Xinje XCPPro project, PLC1: XC3-24 (software 3.3m)

PROGRAM Ladder

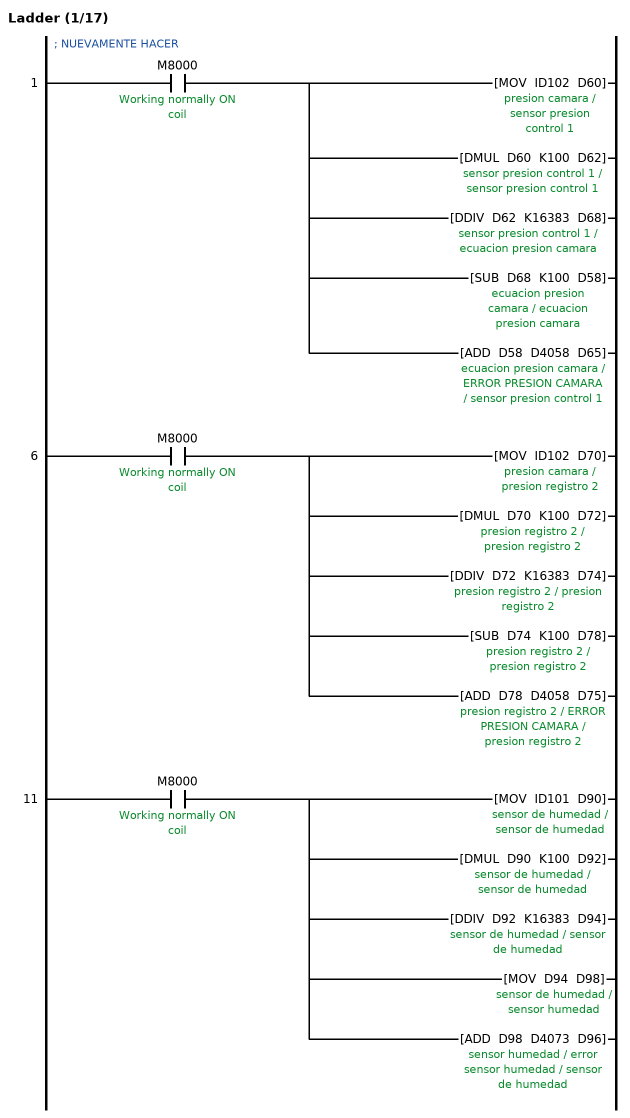
;  NUEVAMENTE HACER
LD     M8000	; Working normally ON coil
MOV    ID102 D60	; presion camara / sensor presion control 1
DMUL   D60 K100 D62	; sensor presion control 1 / sensor presion control 1
DDIV   D62 K16383 D68	; sensor presion control 1 / ecuacion presion camara
SUB    D68 K100 D58	; ecuacion presion camara / ecuacion presion camara
ADD    D58 D4058 D65	; ecuacion presion camara / ERROR PRESION CAMARA / sensor presion control 1
LD     M8000	; Working normally ON coil
MOV    ID102 D70	; presion camara / presion registro 2
DMUL   D70 K100 D72	; presion registro 2 / presion registro 2
DDIV   D72 K16383 D74	; presion registro 2 / presion registro 2
SUB    D74 K100 D78	; presion registro 2 / presion registro 2
ADD    D78 D4058 D75	; presion registro 2 / ERROR PRESION CAMARA / presion registro 2
LD     M8000	; Working normally ON coil
MOV    ID101 D90	; sensor de humedad / sensor de humedad
DMUL   D90 K100 D92	; sensor de humedad / sensor de humedad
DDIV   D92 K16383 D94	; sensor de humedad / sensor de humedad
MOV    D94 D98	; sensor de humedad / sensor humedad
ADD    D98 D4073 D96	; sensor humedad / error sensor humedad / sensor de humedad

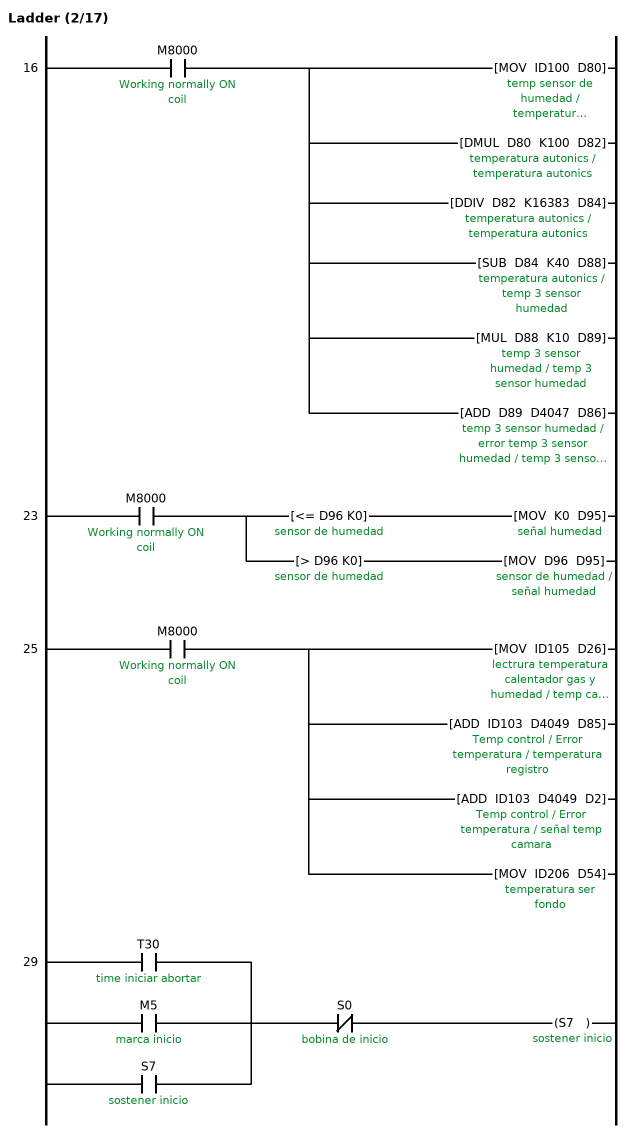
LD     M8000	; Working normally ON coil
MOV    ID100 D80	; temp sensor de humedad / temperatura autonics
DMUL   D80 K100 D82	; temperatura autonics / temperatura autonics
DDIV   D82 K16383 D84	; temperatura autonics / temperatura autonics
SUB    D84 K40 D88	; temperatura autonics / temp 3 sensor humedad
MUL    D88 K10 D89	; temp 3 sensor humedad / temp 3 sensor humedad
ADD    D89 D4047 D86	; temp 3 sensor humedad / error temp 3 sensor humedad / temp 3 sensor humedad
LD     M8000	; Working normally ON coil
MPS
AND<=  D96 K0	; sensor de humedad
MOV    K0 D95	; señal humedad
MPP
AND>   D96 K0	; sensor de humedad
MOV    D96 D95	; sensor de humedad / señal humedad
LD     M8000	; Working normally ON coil
MOV    ID105 D26	; lectrura temperatura  calentador gas y humedad / temp cal gas
ADD    ID103 D4049 D85	; Temp control / Error temperatura / temperatura registro
ADD    ID103 D4049 D2	; Temp control / Error temperatura / señal temp camara
MOV    ID206 D54	; temperatura ser fondo
LD     T30	; time iniciar abortar
OR     M5	; marca inicio
OR     S7	; sostener inicio
ANI    S0	; bobina de inicio
OUT    S7	; sostener inicio

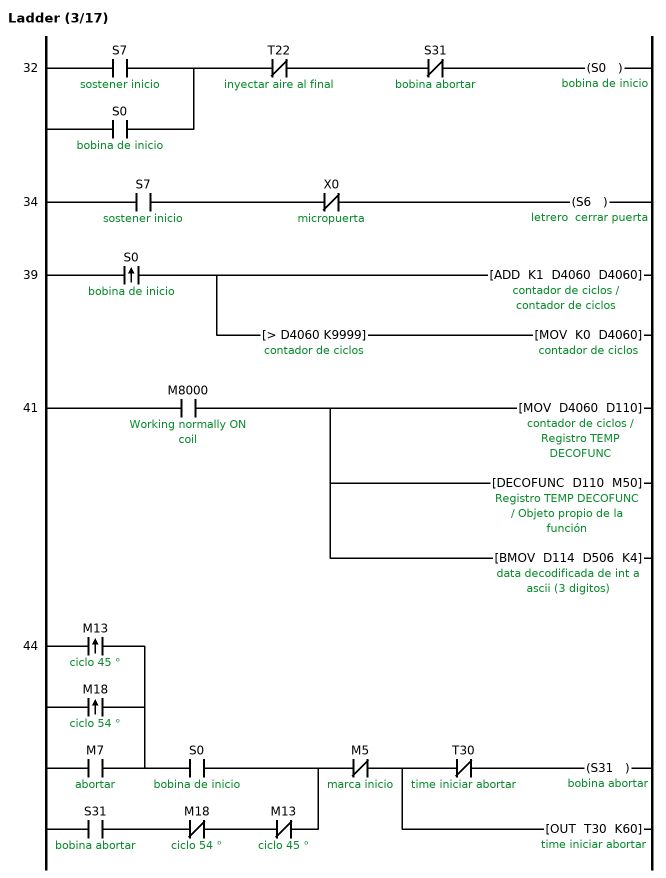
LD     S7	; sostener inicio
OR     S0	; bobina de inicio
ANI    T22	; inyectar aire al final
ANI    S31	; bobina abortar
OUT    S0	; bobina de inicio
LD     S7	; sostener inicio
ANI    X0	;  micropuerta
OUT    S6	; letrero  cerrar puerta
LDP    S0	; bobina de inicio
ADD    K1 D4060 D4060	; contador de ciclos / contador de ciclos
AND>   D4060 K9999	; contador de ciclos
MOV    K0 D4060	; contador de ciclos
LD     M8000	; Working normally ON coil
MOV    D4060 D110	; contador de ciclos / Registro TEMP DECOFUNC
DECOFUNC D110 M50	; Registro TEMP DECOFUNC / Objeto propio de la función
BMOV   D114 D506 K4	; data decodificada de int a ascii (3 digitos)
LDP    M13	; ciclo 45 °
ORP    M18	; ciclo 54 °
OR     M7	; abortar
AND    S0	; bobina de inicio
LD     S31	; bobina abortar
ANI    M18	; ciclo 54 °
ANI    M13	; ciclo 45 °
ORB
ANI    M5	; marca inicio
MPS
ANI    T30	; time iniciar abortar
OUT    S31	; bobina abortar
MPP
OUT    T30 K60	; time iniciar abortar

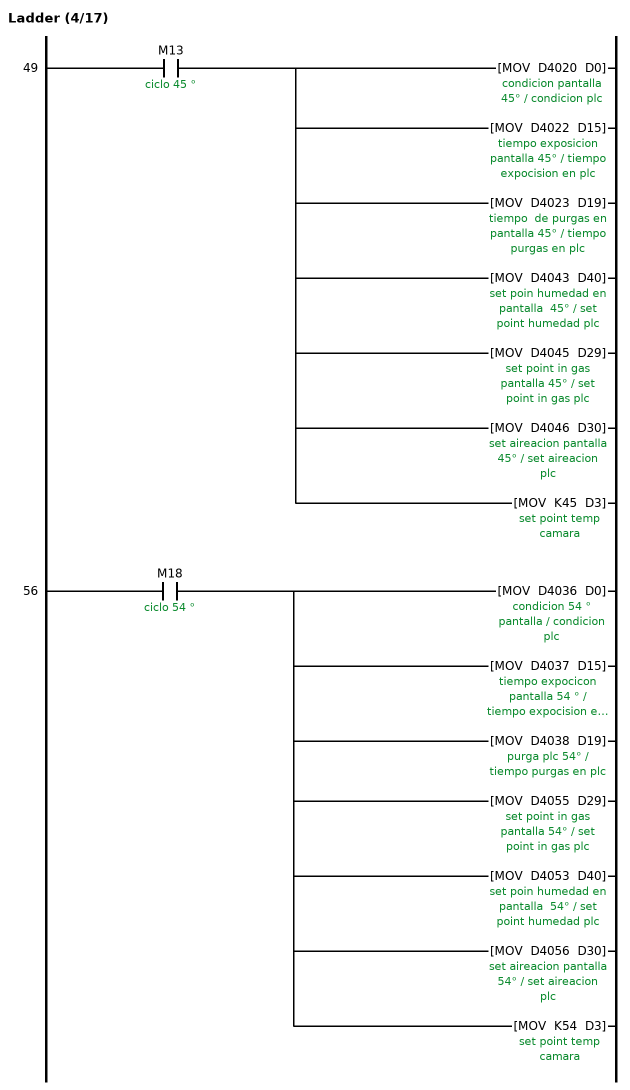
LD     M13	; ciclo 45 °
MOV    D4020 D0	; condicion pantalla 45° / condicion plc
MOV    D4022 D15	; tiempo exposicion pantalla 45° / tiempo expocision en plc
MOV    D4023 D19	; tiempo  de purgas en pantalla 45° / tiempo purgas en plc
MOV    D4043 D40	; set poin humedad en pantalla  45° / set point humedad plc
MOV    D4045 D29	; set point in gas  pantalla 45° / set point in gas plc
MOV    D4046 D30	; set aireacion pantalla 45° / set aireacion plc
MOV    K45 D3	; set point temp camara
LD     M18	; ciclo 54 °
MOV    D4036 D0	; condicion 54 ° pantalla / condicion plc
MOV    D4037 D15	; tiempo expocicon pantalla 54 ° / tiempo expocision en plc
MOV    D4038 D19	; purga plc 54° / tiempo purgas en plc
MOV    D4055 D29	; set point in gas  pantalla 54° / set point in gas plc
MOV    D4053 D40	; set poin humedad en pantalla  54° / set point humedad plc
MOV    D4056 D30	; set aireacion pantalla 54° / set aireacion plc
MOV    K54 D3	; set point temp camara

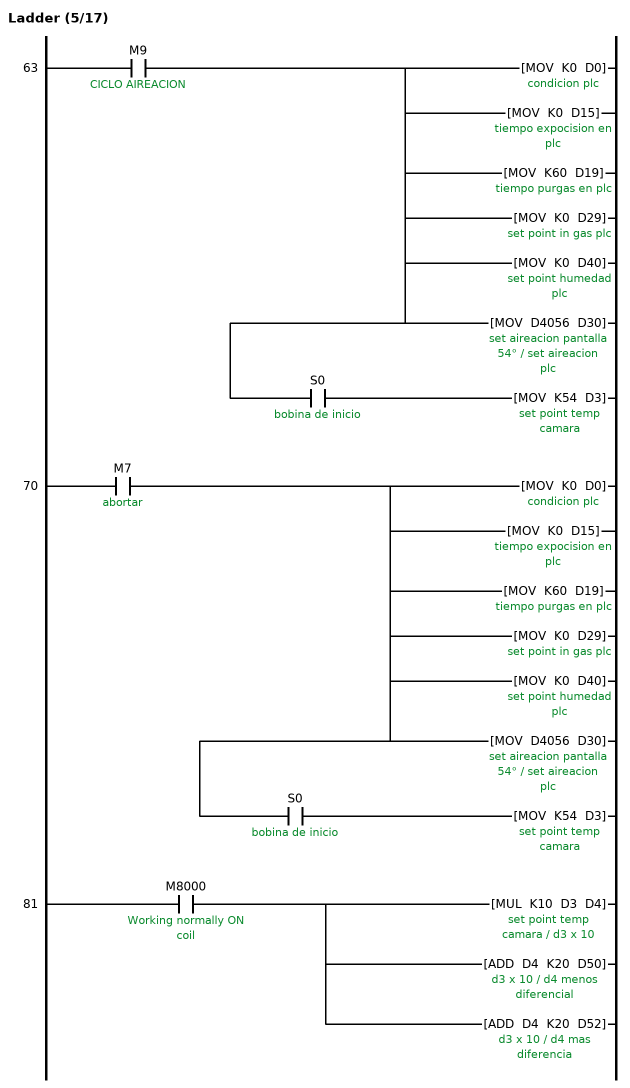
LD     M9	; CICLO AIREACION
MOV    K0 D0	; condicion plc
MOV    K0 D15	; tiempo expocision en plc
MOV    K60 D19	; tiempo purgas en plc
MOV    K0 D29	; set point in gas plc
MOV    K0 D40	; set point humedad plc
MOV    D4056 D30	; set aireacion pantalla 54° / set aireacion plc
AND    S0	; bobina de inicio
MOV    K54 D3	; set point temp camara
LD     M7	; abortar
MOV    K0 D0	; condicion plc
MOV    K0 D15	; tiempo expocision en plc
MOV    K60 D19	; tiempo purgas en plc
MOV    K0 D29	; set point in gas plc
MOV    K0 D40	; set point humedad plc
MOV    D4056 D30	; set aireacion pantalla 54° / set aireacion plc
AND    S0	; bobina de inicio
MOV    K54 D3	; set point temp camara
LD     M8000	; Working normally ON coil
MUL    K10 D3 D4	; set point temp camara / d3 x 10
ADD    D4 K20 D50	; d3 x 10 / d4 menos diferencial
ADD    D4 K20 D52	; d3 x 10 / d4 mas diferencia

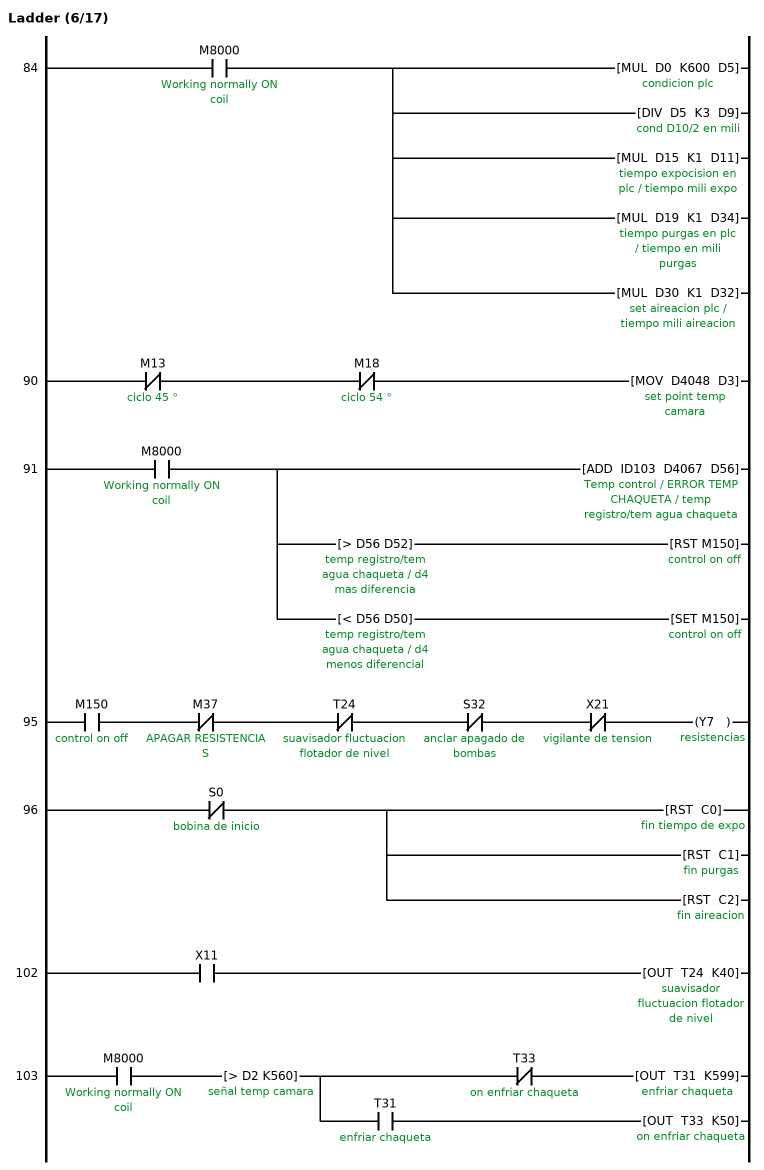
LD     M8000	; Working normally ON coil
MUL    D0 K600 D5	; condicion plc
DIV    D5 K3 D9	; cond D10/2 en mili
MUL    D15 K1 D11	; tiempo expocision en plc / tiempo mili expo
MUL    D19 K1 D34	; tiempo purgas en plc / tiempo en mili purgas
MUL    D30 K1 D32	; set aireacion plc / tiempo mili aireacion
LDI    M13	; ciclo 45 °
ANI    M18	; ciclo 54 °
MOV    D4048 D3	; set point temp camara
LD     M8000	; Working normally ON coil
ADD    ID103 D4067 D56	; Temp control / ERROR TEMP CHAQUETA / temp registro/tem agua chaqueta
MPS
AND>   D56 D52	; temp registro/tem agua chaqueta / d4 mas diferencia
RST    M150	; control on off
MPP
AND<   D56 D50	; temp registro/tem agua chaqueta / d4 menos diferencial
SET    M150	; control on off
LD     M150	; control on off
ANI    M37	; APAGAR RESISTENCIAS
ANI    T24	; suavisador fluctuacion flotador de nivel
ANI    S32	; anclar apagado de bombas
ANI    X21	; vigilante de tension
OUT    Y7	; resistencias
LDI    S0	; bobina de inicio
RST    C0	; fin tiempo de expo
RST    C1	; fin purgas
RST    C2	; fin aireacion
LD     X11
OUT    T24 K40	; suavisador fluctuacion flotador de nivel
LD     M8000	; Working normally ON coil
AND>   D2 K560	; señal temp camara
MPS
ANI    T33	; on enfriar chaqueta
OUT    T31 K599	; enfriar chaqueta
MPP
AND    T31	; enfriar chaqueta
OUT    T33 K50	; on enfriar chaqueta

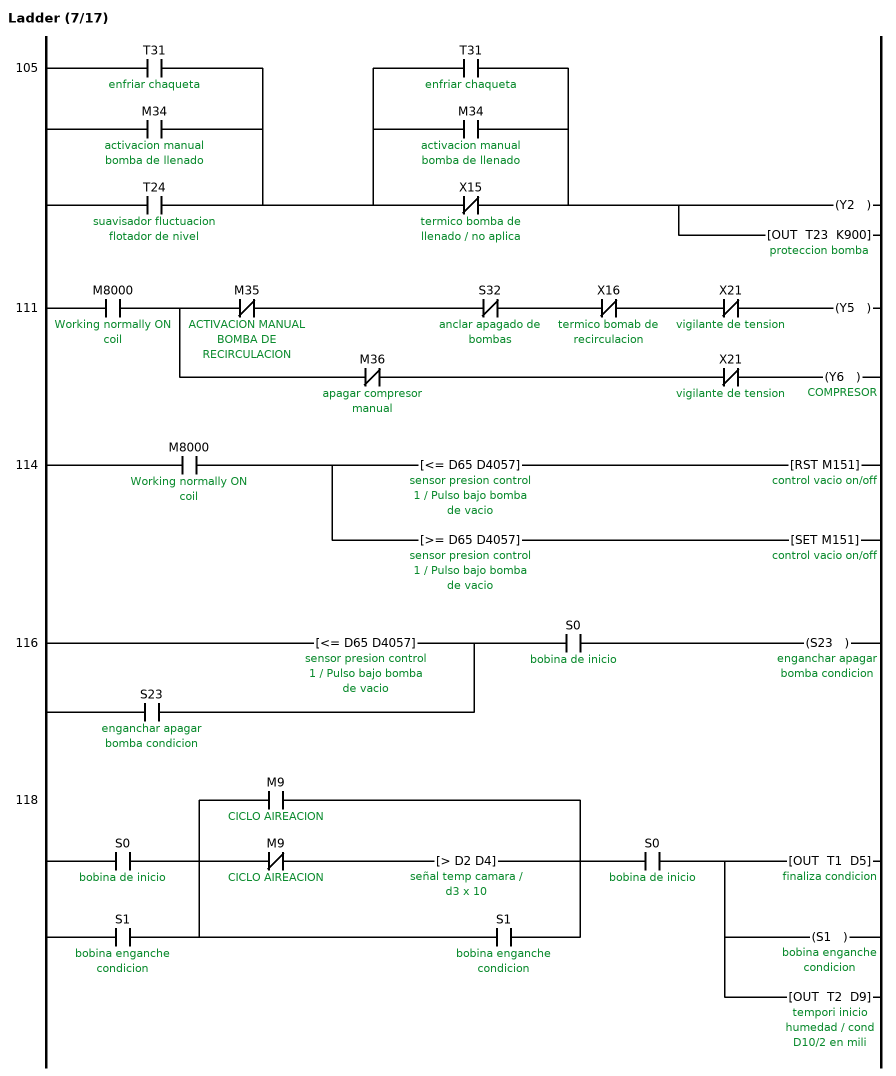
LD     T31	; enfriar chaqueta
OR     M34	; activacion manual bomba de llenado
OR     T24	; suavisador fluctuacion flotador de nivel
LD     T31	; enfriar chaqueta
OR     M34	; activacion manual bomba de llenado
ORI    X15	; termico bomba de  llenado / no aplica 
ANB
OUT    Y2
OUT    T23 K900	; proteccion bomba
LD     M8000	; Working normally ON coil
MPS
ANI    M35	; ACTIVACION MANUAL BOMBA DE RECIRCULACION
ANI    S32	; anclar apagado de bombas
ANI    X16	; termico bomab de recirculacion
ANI    X21	; vigilante de tension
OUT    Y5
MPP
ANI    M36	; apagar compresor manual
ANI    X21	; vigilante de tension
OUT    Y6	; COMPRESOR
LD     M8000	; Working normally ON coil
MPS
AND<=  D65 D4057	; sensor presion control 1 / Pulso bajo bomba de vacio
RST    M151	; control vacio on/off
MPP
AND>=  D65 D4057	; sensor presion control 1 / Pulso bajo bomba de vacio
SET    M151	; control vacio on/off
LD<=   D65 D4057	; sensor presion control 1 / Pulso bajo bomba de vacio
OR     S23	; enganchar apagar bomba condicion
AND    S0	; bobina de inicio
OUT    S23	; enganchar apagar bomba condicion
LD     S0	; bobina de inicio
OR     S1	; bobina enganche  condicion
LD     M9	; CICLO AIREACION
LDI    M9	; CICLO AIREACION
AND>   D2 D4	; señal temp camara / d3 x 10
ORB
OR     S1	; bobina enganche  condicion
ANB
AND    S0	; bobina de inicio
OUT    T1 D5	; finaliza condicion
OUT    S1	; bobina enganche  condicion
OUT    T2 D9	; tempori inicio humedad / cond D10/2 en mili

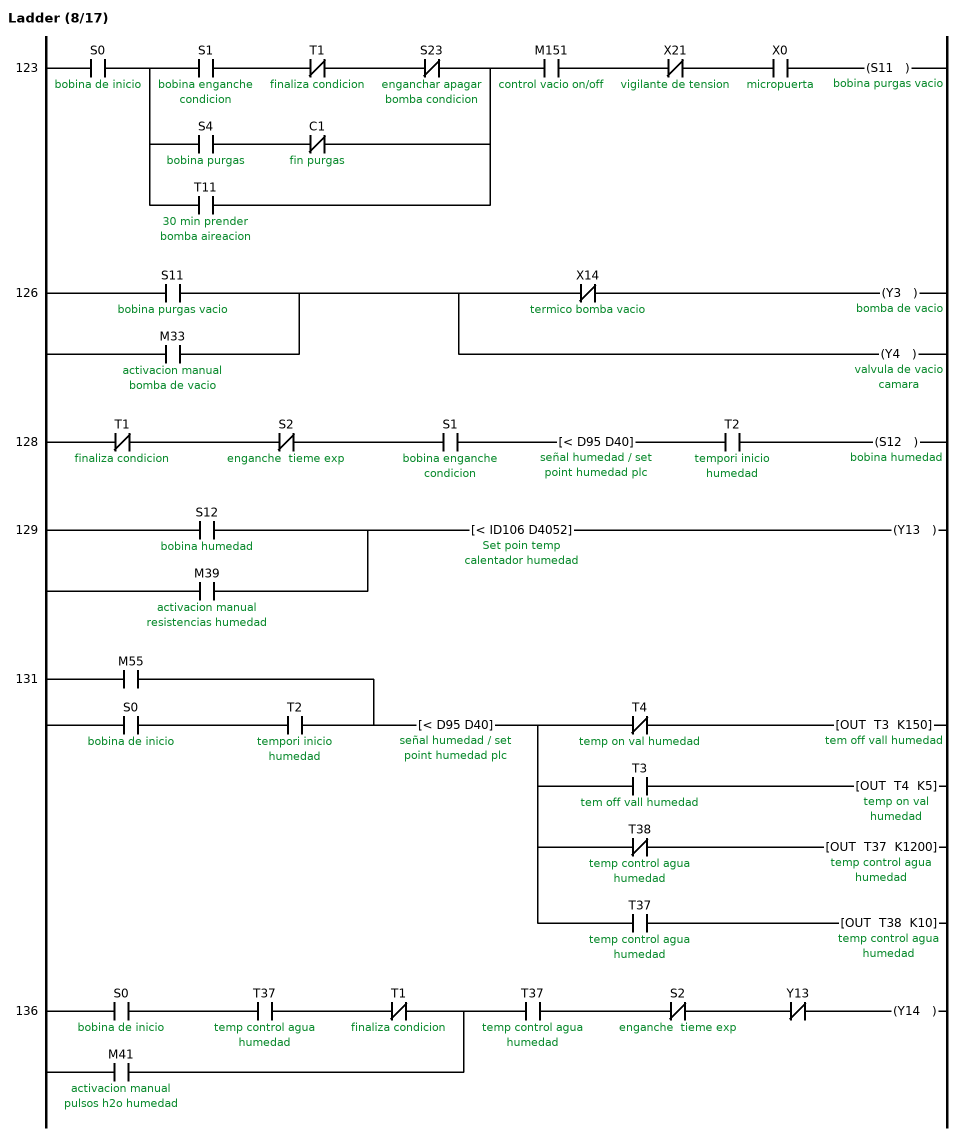
LD     S0	; bobina de inicio
LD     S1	; bobina enganche  condicion
ANI    T1	; finaliza condicion
ANI    S23	; enganchar apagar bomba condicion
LD     S4	; bobina purgas
ANI    C1	; fin purgas
ORB
OR     T11	; 30 min prender bomba aireacion
ANB
AND    M151	; control vacio on/off
ANI    X21	; vigilante de tension
AND    X0	;  micropuerta
OUT    S11	; bobina purgas vacio
LD     S11	; bobina purgas vacio
OR     M33	; activacion manual bomba de vacio
MPS
ANI    X14	; termico bomba vacio
OUT    Y3	; bomba de vacio
MPP
OUT    Y4	; valvula de vacio camara
LDI    T1	; finaliza condicion
ANI    S2	; enganche  tieme exp
AND    S1	; bobina enganche  condicion
AND<   D95 D40	; señal humedad / set point humedad plc
AND    T2	; tempori inicio humedad
OUT    S12	; bobina humedad
LD     S12	; bobina humedad
OR     M39	; activacion manual resistencias humedad
AND<   ID106 D4052	; Set poin temp calentador humedad
OUT    Y13
LD     M55
LD     S0	; bobina de inicio
AND    T2	; tempori inicio humedad
ORB
AND<   D95 D40	; señal humedad / set point humedad plc
MPS
ANI    T4	; temp on val humedad
OUT    T3 K150	; tem off vall humedad
MRD
AND    T3	; tem off vall humedad
OUT    T4 K5	; temp on val humedad
MRD
ANI    T38	; temp control agua humedad
OUT    T37 K1200	; temp control agua  humedad
MPP
AND    T37	; temp control agua  humedad
OUT    T38 K10	; temp control agua humedad
LD     S0	; bobina de inicio
AND    T37	; temp control agua  humedad
ANI    T1	; finaliza condicion
OR     M41	; activacion manual pulsos h2o humedad
AND    T37	; temp control agua  humedad
ANI    S2	; enganche  tieme exp
ANI    Y13
OUT    Y14

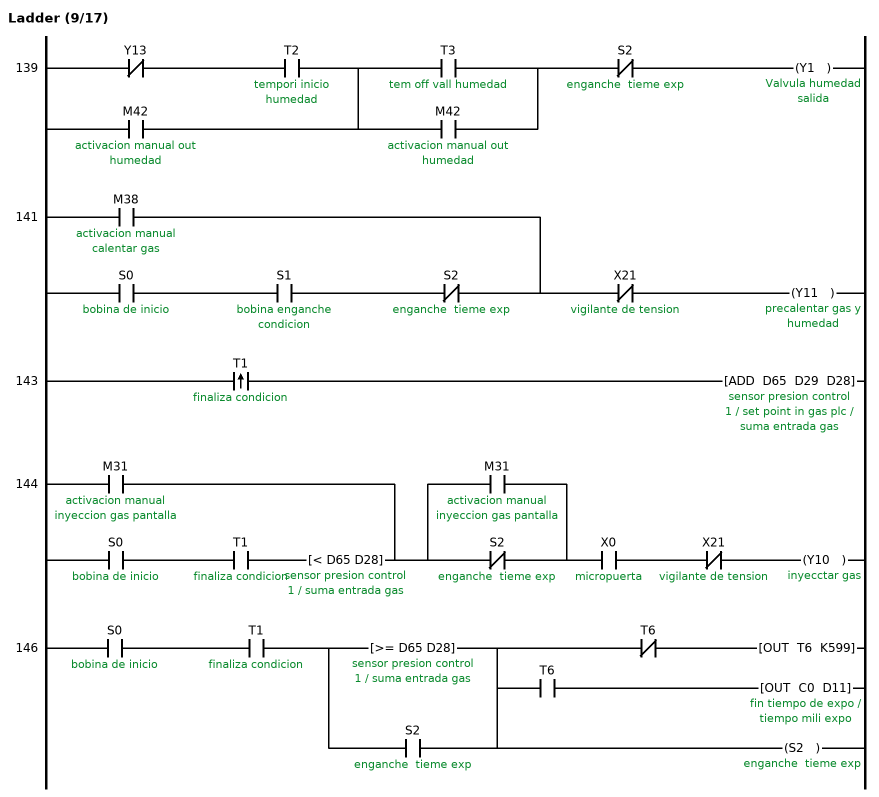
LDI    Y13
AND    T2	; tempori inicio humedad
OR     M42	; activacion manual out humedad
LD     T3	; tem off vall humedad
OR     M42	; activacion manual out humedad
ANB
ANI    S2	; enganche  tieme exp
OUT    Y1	; Valvula humedad salida
LD     M38	; activacion manual calentar gas
LD     S0	; bobina de inicio
AND    S1	; bobina enganche  condicion
ANI    S2	; enganche  tieme exp
ORB
ANI    X21	; vigilante de tension
OUT    Y11	; precalentar gas y humedad
LDP    T1	; finaliza condicion
ADD    D65 D29 D28	; sensor presion control 1 / set point in gas plc / suma entrada gas
LD     M31	; activacion manual inyeccion gas pantalla
LD     S0	; bobina de inicio
AND    T1	; finaliza condicion
AND<   D65 D28	; sensor presion control 1 / suma entrada gas
ORB
LD     M31	; activacion manual inyeccion gas pantalla
ORI    S2	; enganche  tieme exp
ANB
AND    X0	;  micropuerta
ANI    X21	; vigilante de tension
OUT    Y10	; inyecctar gas
LD     S0	; bobina de inicio
AND    T1	; finaliza condicion
LD>=   D65 D28	; sensor presion control 1 / suma entrada gas
OR     S2	; enganche  tieme exp
ANB
MPS
ANI    T6
OUT    T6 K599
MRD
AND    T6
OUT    C0 D11	; fin tiempo de expo / tiempo mili expo
MPP
OUT    S2	; enganche  tieme exp

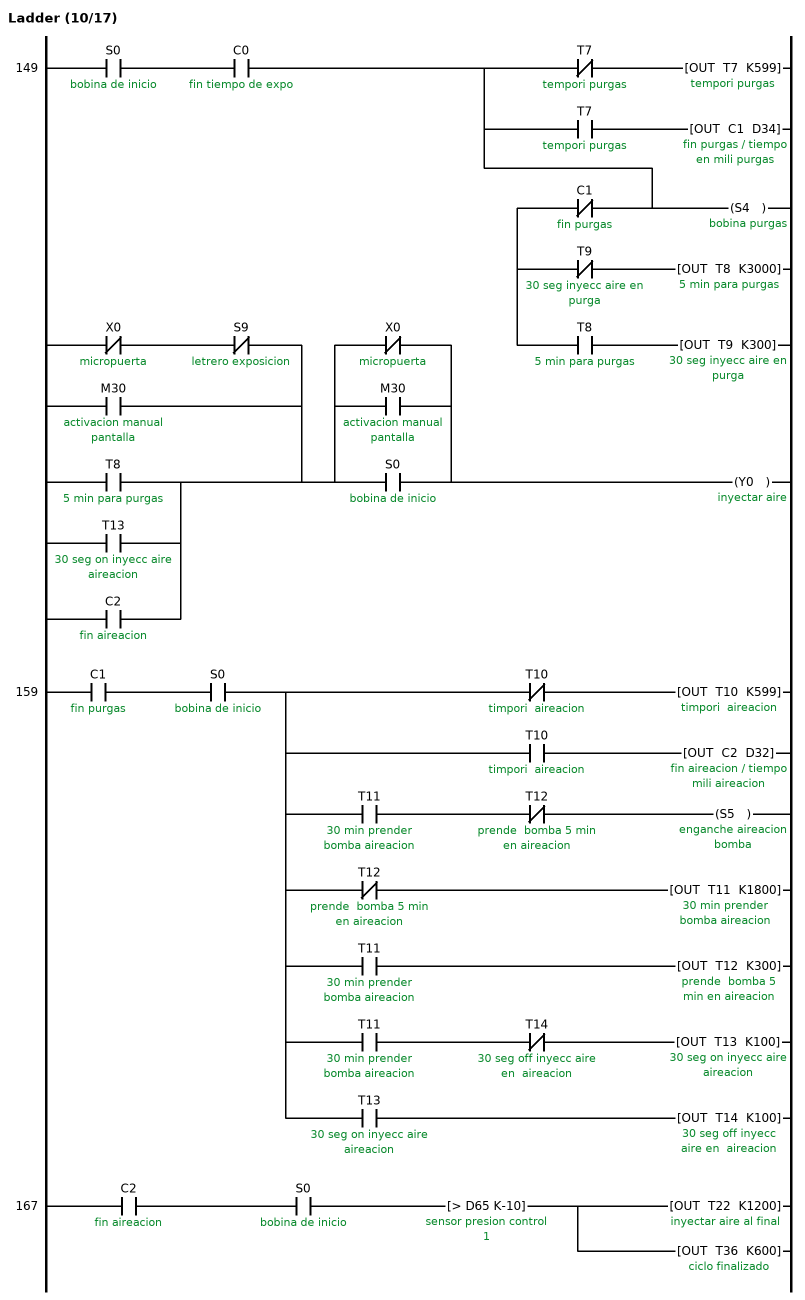
; (network is not series-parallel: see picture) LD S0 | LD C0 | LDI T7 | OUT T7 K599 | LD T7 | OUT C1 D34 | LDI C1 | OUT S4 | LDI T9 | OUT T8 K3000 | LDI X0 | LDI S9 | LDI X0 | LD T8 | OUT T9 K300 | LD M30 | LD M30 | LD T8 | LD S0 | OUT Y0 | LD T13 | LD C2
LD     C1	; fin purgas
AND    S0	; bobina de inicio
MPS
ANI    T10	; timpori  aireacion
OUT    T10 K599	; timpori  aireacion
MRD
AND    T10	; timpori  aireacion
OUT    C2 D32	; fin aireacion / tiempo mili aireacion
MRD
AND    T11	; 30 min prender bomba aireacion
ANI    T12	; prende  bomba 5 min en aireacion
OUT    S5	; enganche aireacion bomba
MRD
ANI    T12	; prende  bomba 5 min en aireacion
OUT    T11 K1800	; 30 min prender bomba aireacion
MRD
AND    T11	; 30 min prender bomba aireacion
OUT    T12 K300	; prende  bomba 5 min en aireacion
MRD
AND    T11	; 30 min prender bomba aireacion
ANI    T14	; 30 seg off inyecc aire en  aireacion
OUT    T13 K100	; 30 seg on inyecc aire aireacion
MPP
AND    T13	; 30 seg on inyecc aire aireacion
OUT    T14 K100	; 30 seg off inyecc aire en  aireacion
LD     C2	; fin aireacion
AND    S0	; bobina de inicio
AND>   D65 K-10	; sensor presion control 1
OUT    T22 K1200	; inyectar aire al final
OUT    T36 K600	; ciclo finalizado

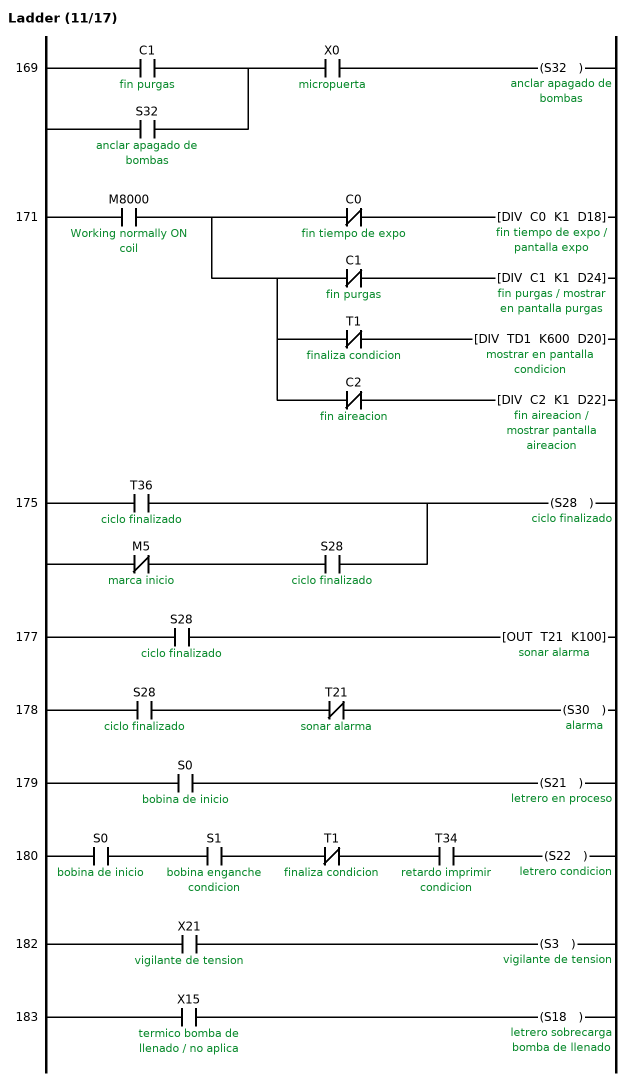
LD     C1	; fin purgas
OR     S32	; anclar apagado de bombas
AND    X0	;  micropuerta
OUT    S32	; anclar apagado de bombas
LD     M8000	; Working normally ON coil
MPS
ANI    C0	; fin tiempo de expo
DIV    C0 K1 D18	; fin tiempo de expo / pantalla expo
MRD
ANI    C1	; fin purgas
DIV    C1 K1 D24	; fin purgas / mostrar en pantalla purgas
MRD
ANI    T1	; finaliza condicion
DIV    TD1 K600 D20	; mostrar en pantalla condicion
MPP
ANI    C2	; fin aireacion
DIV    C2 K1 D22	; fin aireacion / mostrar pantalla aireacion
LD     T36	; ciclo finalizado
LDI    M5	; marca inicio
AND    S28	; ciclo finalizado
ORB
OUT    S28	; ciclo finalizado
LD     S28	; ciclo finalizado
OUT    T21 K100	; sonar alarma
LD     S28	; ciclo finalizado
ANI    T21	; sonar alarma
OUT    S30	; alarma
LD     S0	; bobina de inicio
OUT    S21	; letrero en proceso
LD     S0	; bobina de inicio
AND    S1	; bobina enganche  condicion
ANI    T1	; finaliza condicion
AND    T34	; retardo imprimir condicion
OUT    S22	; letrero condicion
LD     X21	; vigilante de tension
OUT    S3	; vigilante de tension
LD     X15	; termico bomba de  llenado / no aplica 
OUT    S18	; letrero sobrecarga bomba de llenado

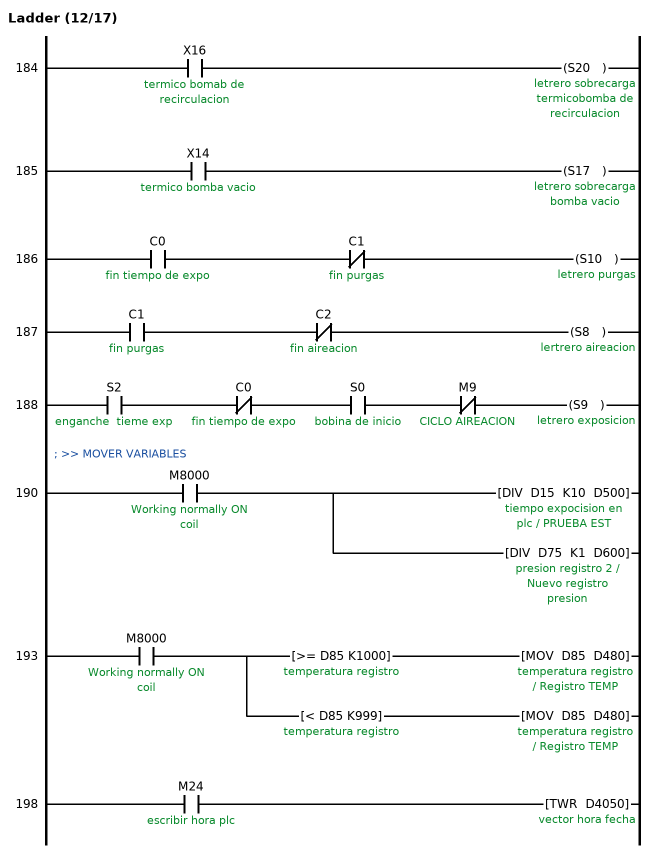
LD     X16	; termico bomab de recirculacion
OUT    S20	; letrero sobrecarga termicobomba de recirculacion
LD     X14	; termico bomba vacio
OUT    S17	; letrero sobrecarga bomba vacio
LD     C0	; fin tiempo de expo
ANI    C1	; fin purgas
OUT    S10	; letrero purgas
LD     C1	; fin purgas
ANI    C2	; fin aireacion
OUT    S8	; lertrero aireacion
LD     S2	; enganche  tieme exp
ANI    C0	; fin tiempo de expo
AND    S0	; bobina de inicio
ANI    M9	; CICLO AIREACION
OUT    S9	; letrero exposicion
;  >> MOVER VARIABLES
LD     M8000	; Working normally ON coil
DIV    D15 K10 D500	; tiempo expocision en plc / PRUEBA EST
DIV    D75 K1 D600	; presion registro 2 / Nuevo registro presion 
LD     M8000	; Working normally ON coil
MPS
AND>=  D85 K1000	; temperatura registro
MOV    D85 D480	; temperatura registro / Registro TEMP 
MPP
AND<   D85 K999	; temperatura registro
MOV    D85 D480	; temperatura registro / Registro TEMP 
LD     M24	; escribir hora plc
TWR    D4050	; vector hora fecha

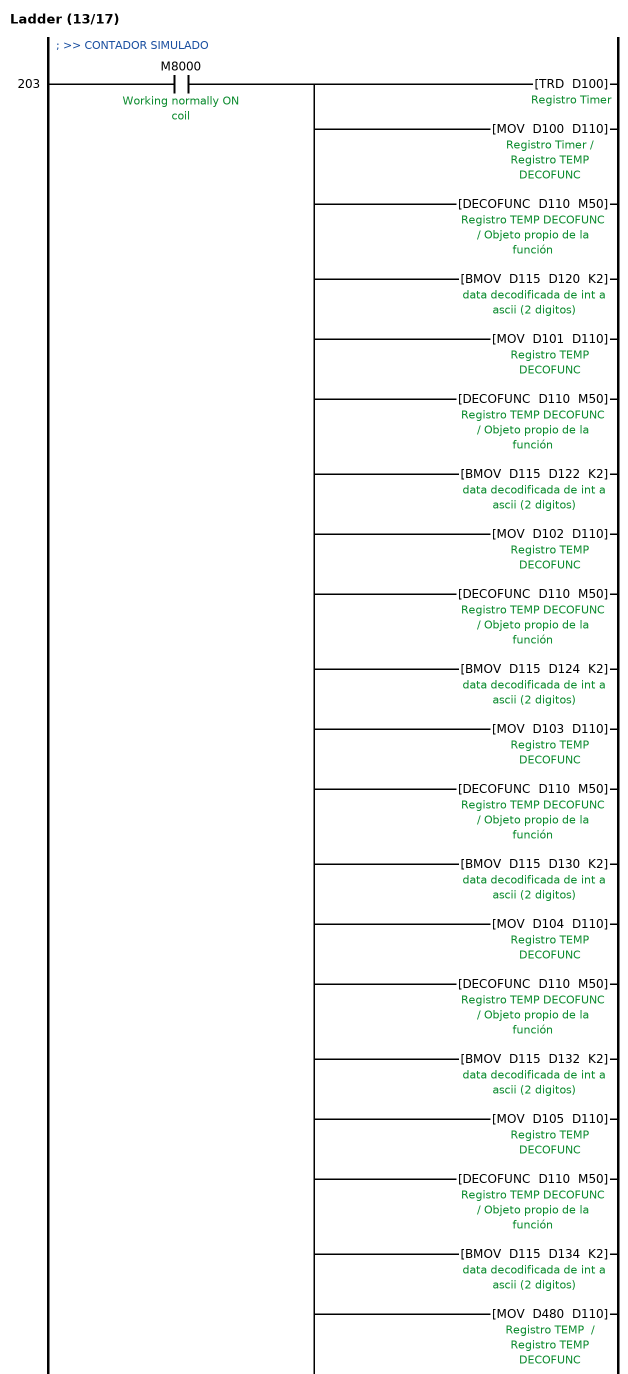
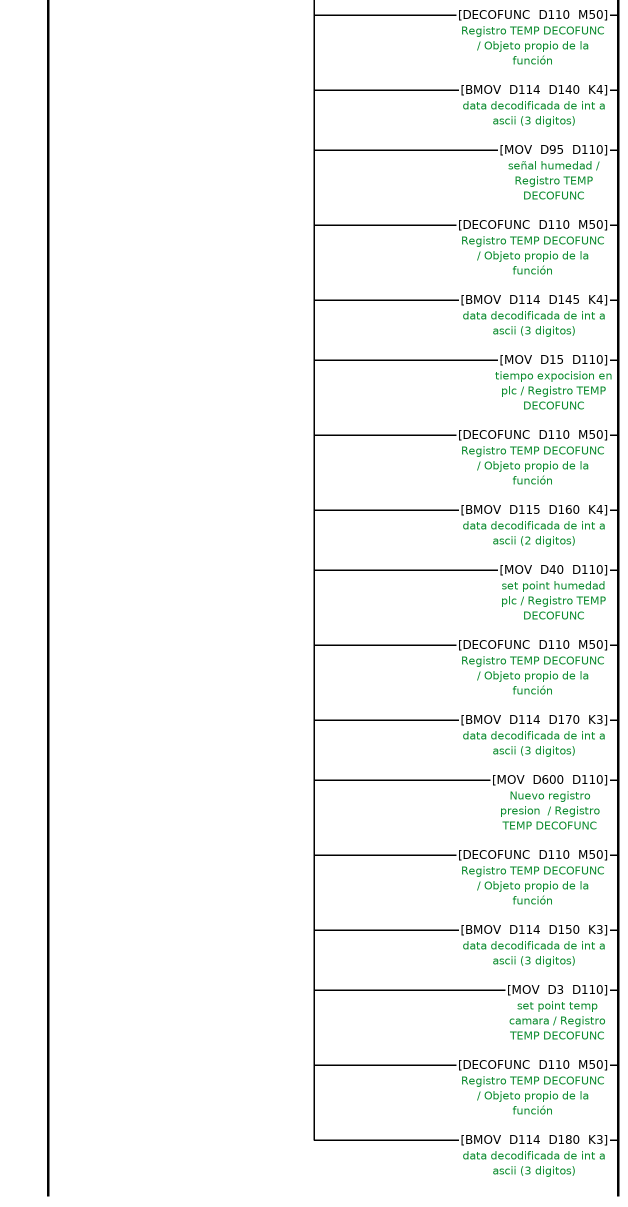
; >> CONTADOR SIMULADO
LD     M8000	; Working normally ON coil
TRD    D100	; Registro Timer
MOV    D100 D110	; Registro Timer / Registro TEMP DECOFUNC
DECOFUNC D110 M50	; Registro TEMP DECOFUNC / Objeto propio de la función
BMOV   D115 D120 K2	; data decodificada de int a ascii (2 digitos)
MOV    D101 D110	; Registro TEMP DECOFUNC
DECOFUNC D110 M50	; Registro TEMP DECOFUNC / Objeto propio de la función
BMOV   D115 D122 K2	; data decodificada de int a ascii (2 digitos)
MOV    D102 D110	; Registro TEMP DECOFUNC
DECOFUNC D110 M50	; Registro TEMP DECOFUNC / Objeto propio de la función
BMOV   D115 D124 K2	; data decodificada de int a ascii (2 digitos)
MOV    D103 D110	; Registro TEMP DECOFUNC
DECOFUNC D110 M50	; Registro TEMP DECOFUNC / Objeto propio de la función
BMOV   D115 D130 K2	; data decodificada de int a ascii (2 digitos)
MOV    D104 D110	; Registro TEMP DECOFUNC
DECOFUNC D110 M50	; Registro TEMP DECOFUNC / Objeto propio de la función
BMOV   D115 D132 K2	; data decodificada de int a ascii (2 digitos)
MOV    D105 D110	; Registro TEMP DECOFUNC
DECOFUNC D110 M50	; Registro TEMP DECOFUNC / Objeto propio de la función
BMOV   D115 D134 K2	; data decodificada de int a ascii (2 digitos)
MOV    D480 D110	; Registro TEMP  / Registro TEMP DECOFUNC
DECOFUNC D110 M50	; Registro TEMP DECOFUNC / Objeto propio de la función
BMOV   D114 D140 K4	; data decodificada de int a ascii (3 digitos)
MOV    D95 D110	; señal humedad / Registro TEMP DECOFUNC
DECOFUNC D110 M50	; Registro TEMP DECOFUNC / Objeto propio de la función
BMOV   D114 D145 K4	; data decodificada de int a ascii (3 digitos)
MOV    D15 D110	; tiempo expocision en plc / Registro TEMP DECOFUNC
DECOFUNC D110 M50	; Registro TEMP DECOFUNC / Objeto propio de la función
BMOV   D115 D160 K4	; data decodificada de int a ascii (2 digitos)
MOV    D40 D110	; set point humedad plc / Registro TEMP DECOFUNC
DECOFUNC D110 M50	; Registro TEMP DECOFUNC / Objeto propio de la función
BMOV   D114 D170 K3	; data decodificada de int a ascii (3 digitos)
MOV    D600 D110	; Nuevo registro presion  / Registro TEMP DECOFUNC
DECOFUNC D110 M50	; Registro TEMP DECOFUNC / Objeto propio de la función
BMOV   D114 D150 K3	; data decodificada de int a ascii (3 digitos)
MOV    D3 D110	; set point temp camara / Registro TEMP DECOFUNC
DECOFUNC D110 M50	; Registro TEMP DECOFUNC / Objeto propio de la función
BMOV   D114 D180 K3	; data decodificada de int a ascii (3 digitos)

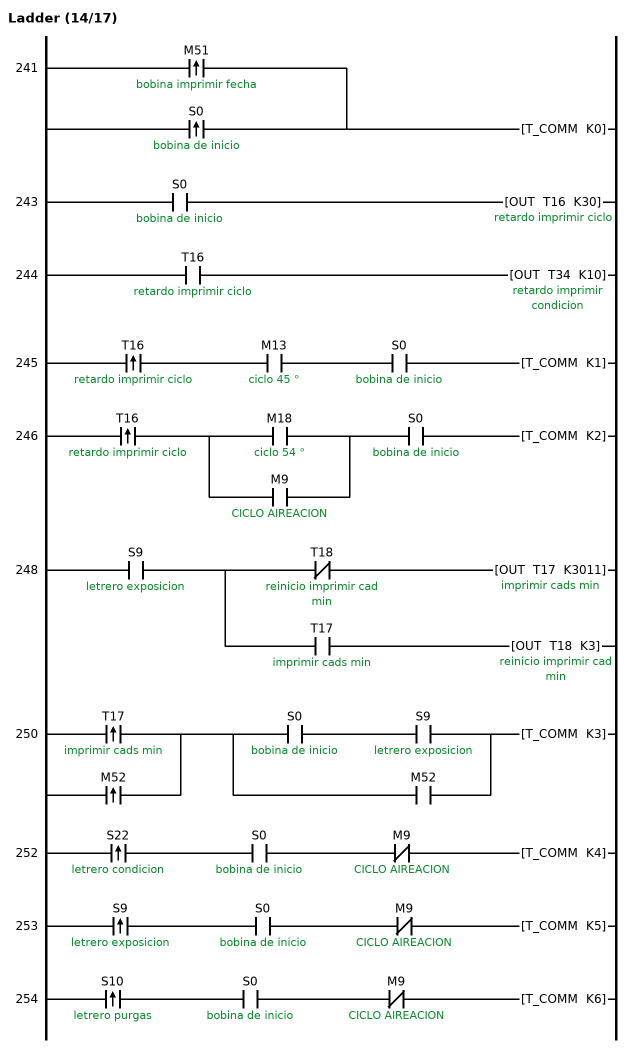
LDP    M51	; bobina imprimir fecha
ORP    S0	; bobina de inicio
T_COMM K0
LD     S0	; bobina de inicio
OUT    T16 K30	; retardo imprimir ciclo
LD     T16	; retardo imprimir ciclo
OUT    T34 K10	; retardo imprimir condicion
LDP    T16	; retardo imprimir ciclo
AND    M13	; ciclo 45 °
AND    S0	; bobina de inicio
T_COMM K1
LDP    T16	; retardo imprimir ciclo
LD     M18	; ciclo 54 °
OR     M9	; CICLO AIREACION
ANB
AND    S0	; bobina de inicio
T_COMM K2
LD     S9	; letrero exposicion
MPS
ANI    T18	; reinicio imprimir cad min
OUT    T17 K3011	; imprimir cads min
MPP
AND    T17	; imprimir cads min
OUT    T18 K3	; reinicio imprimir cad min
LDP    T17	; imprimir cads min
ORP    M52
LD     S0	; bobina de inicio
AND    S9	; letrero exposicion
OR     M52
ANB
T_COMM K3
LDP    S22	; letrero condicion
AND    S0	; bobina de inicio
ANI    M9	; CICLO AIREACION
T_COMM K4
LDP    S9	; letrero exposicion
AND    S0	; bobina de inicio
ANI    M9	; CICLO AIREACION
T_COMM K5
LDP    S10	; letrero purgas
AND    S0	; bobina de inicio
ANI    M9	; CICLO AIREACION
T_COMM K6

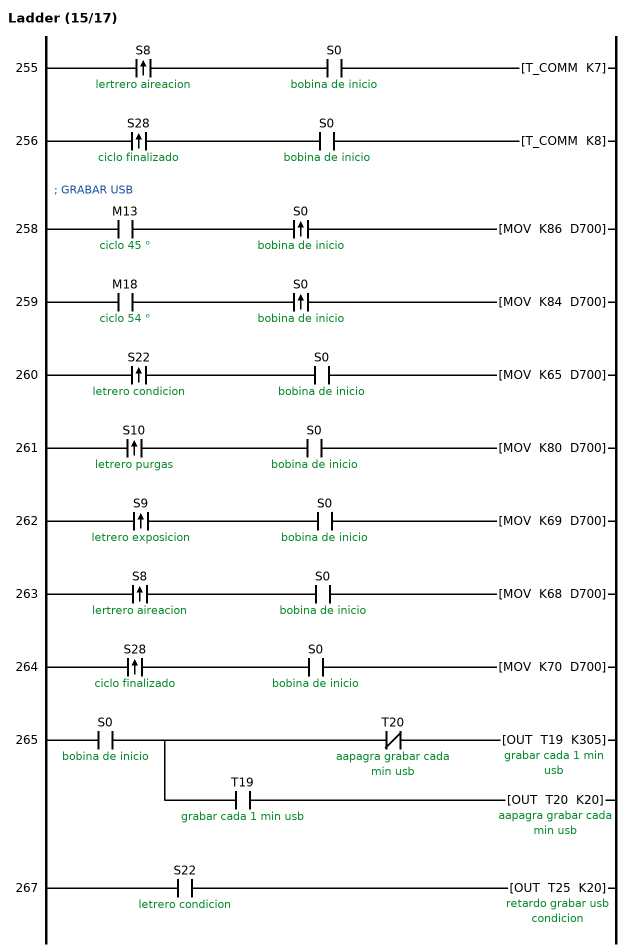
LDP    S8	; lertrero aireacion
AND    S0	; bobina de inicio
T_COMM K7
LDP    S28	; ciclo finalizado
AND    S0	; bobina de inicio
T_COMM K8
;  GRABAR USB
LD     M13	; ciclo 45 °
ANDP   S0	; bobina de inicio
MOV    K86 D700
LD     M18	; ciclo 54 °
ANDP   S0	; bobina de inicio
MOV    K84 D700
LDP    S22	; letrero condicion
AND    S0	; bobina de inicio
MOV    K65 D700
LDP    S10	; letrero purgas
AND    S0	; bobina de inicio
MOV    K80 D700
LDP    S9	; letrero exposicion
AND    S0	; bobina de inicio
MOV    K69 D700
LDP    S8	; lertrero aireacion
AND    S0	; bobina de inicio
MOV    K68 D700
LDP    S28	; ciclo finalizado
AND    S0	; bobina de inicio
MOV    K70 D700
LD     S0	; bobina de inicio
MPS
ANI    T20	; aapagra grabar cada min usb
OUT    T19 K305	; grabar cada 1 min usb
MPP
AND    T19	; grabar cada 1 min usb
OUT    T20 K20	; aapagra grabar cada min usb
LD     S22	; letrero condicion
OUT    T25 K20	; retardo grabar usb condicion

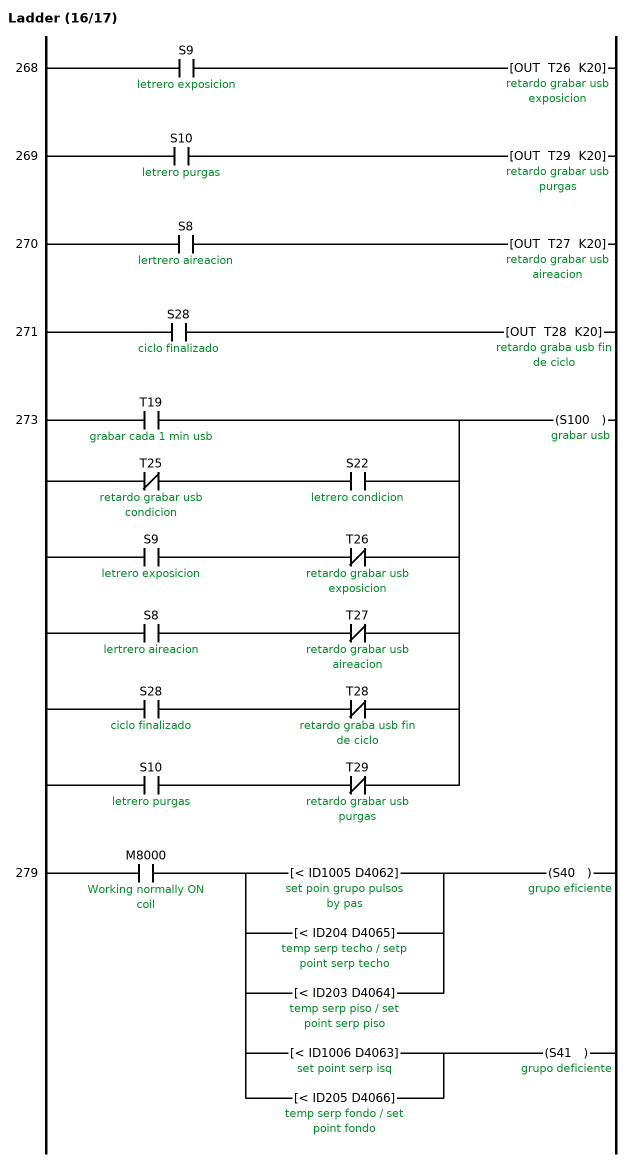
LD     S9	; letrero exposicion
OUT    T26 K20	; retardo grabar usb exposicion
LD     S10	; letrero purgas
OUT    T29 K20	; retardo grabar usb purgas
LD     S8	; lertrero aireacion
OUT    T27 K20	; retardo grabar usb aireacion
LD     S28	; ciclo finalizado
OUT    T28 K20	; retardo graba usb fin de ciclo
LD     T19	; grabar cada 1 min usb
LDI    T25	; retardo grabar usb condicion
AND    S22	; letrero condicion
ORB
LD     S9	; letrero exposicion
ANI    T26	; retardo grabar usb exposicion
ORB
LD     S8	; lertrero aireacion
ANI    T27	; retardo grabar usb aireacion
ORB
LD     S28	; ciclo finalizado
ANI    T28	; retardo graba usb fin de ciclo
ORB
LD     S10	; letrero purgas
ANI    T29	; retardo grabar usb purgas
ORB
OUT    S100	; grabar usb
LD     M8000	; Working normally ON coil
MPS
LD<    ID1005 D4062	; set poin grupo pulsos by pas
OR<    ID204 D4065	; temp serp techo / setp point serp techo
OR<    ID203 D4064	; temp serp piso / set point serp piso
ANB
OUT    S40	; grupo eficiente 
MPP
LD<    ID1006 D4063	; set point serp isq
OR<    ID205 D4066	; temp serp fondo / set point fondo
ANB
OUT    S41	; grupo deficiente

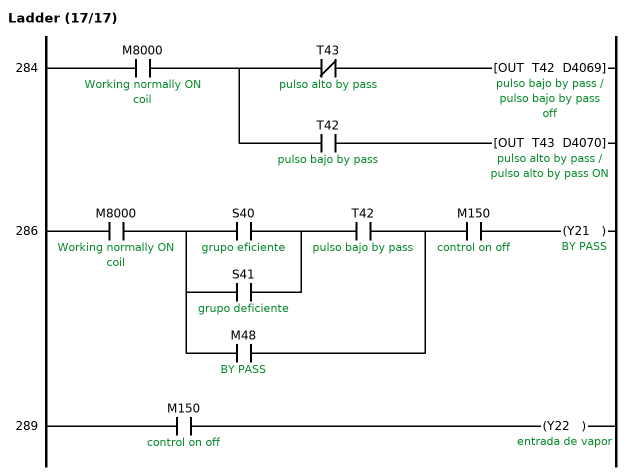
LD     M8000	; Working normally ON coil
MPS
ANI    T43	; pulso alto by pass
OUT    T42 D4069	; pulso bajo by pass / pulso bajo by pass off
MPP
AND    T42	; pulso bajo by pass
OUT    T43 D4070	; pulso alto by pass / pulso alto by pass ON
LD     M8000	; Working normally ON coil
LD     S40	; grupo eficiente 
OR     S41	; grupo deficiente
AND    T42	; pulso bajo by pass
OR     M48	; BY PASS
ANB
AND    M150	; control on off
OUT    Y21	; BY PASS
LD     M150	; control on off
OUT    Y22	; entrada de vapor

COMMENTS (devices not used above)
M43	activar manual hmi der
M44	activar manual hmi sep izq
M45	activar manual hmi sep piso
M46	activar manual hmi sep techo
M47	activar manual hmi sep fondo
S19	letrero  resistencias gas
T15	tempor imprimir fecha
T32	CONTROL DE NIVEL
T44	pulso OFF
T45	pulso on
C3	CONTADOR NIVEL
D10	t mili condicion plc
D12	tiempo en mili purgas
D13	señal temp calen gas
D21	mostrar en pantalla expo
D33	tiempo en mili purgas
D42	contador de ciclos
D61	sensor presion control 1
D63	sensor presion control 1
D64	sensor presion control 1
D71	presion registro 2
D73	presion registro 2
D81	temperatura autonics
D83	temperatura autonics
D91	d80 div 16383
D93	d92 x 9580
D4019	atm presion camara
D4044	set point cal gas pantalla
D4051	Error temp registro
D4071	grupo deficiente sepentin OFF
D4072	grupo eficiente serpentin ON
D4074	temp de inicio
ID1000	lectura sensor de presion
ID1001	lectura puerto humedad HIH 4000
ID1003	lectrura temperatura  camara

CONFIG BLOCK T_COMM K0	; Encabezado
  IsUserInst=false, Inst=SEND, PLCAddr=D1000, ComNum=K2, BufferCount=8, Type=Const, Data="FECHA: ", RegByteCount=0, Type=Reg, Reg=D124, RegByteCount=1, Type=Reg, Reg=D125, RegByteCount=1, Type=Const, Data="/", RegByteCount=0, Type=Reg, Reg=D122, RegByteCount=1, Type=Reg, Reg=D123, RegByteCount=1, Type=Const, Data="/", RegByteCount=0, Type=Reg, Reg=D120, RegByteCount=1, Type=Reg, Reg=D121, RegByteCount=1, Type=Const, Data=13, RegByteCount=0, Type=Const, Data="HORA INICIO: ", RegByteCount=0, Type=Reg, Reg=D130, RegByteCount=1, Type=Reg, Reg=D131, RegByteCount=1, Type=Const, Data=":", RegByteCount=0, Type=Reg, Reg=D132, RegByteCount=1, Type=Reg, Reg=D133, RegByteCount=1, Type=Const, Data=":", RegByteCount=0, Type=Reg, Reg=D134, RegByteCount=1

CONFIG BLOCK T_COMM K1	; Ciclo 45
  IsUserInst=false, Inst=SEND, PLCAddr=D1100, ComNum=K2, BufferCount=8, Type=Const, Data=62, RegByteCount=0, Type=Const, Data=62, RegByteCount=0, Type=Const, Data="CICLO 45", RegByteCount=0, Type=Const, Data=248, RegByteCount=0, Type=Const, Data="C", RegByteCount=0, Type=Const, Data=60, RegByteCount=0, Type=Const, Data=60, RegByteCount=0, Type=Const, Data=13, RegByteCount=0, Type=Const, Data="TEMP:", RegByteCount=0, Type=Reg, Reg=D180, RegByteCount=1, Type=Reg, Reg=D181, RegByteCount=1, Type=Reg, Reg=D182, RegByteCount=1, Type=Const, Data=248, RegByteCount=0, Type=Const, Data=67, RegByteCount=0, Type=Const, Data=32, RegByteCount=0, Type=Const, Data="EXP:", RegByteCount=0, Type=Reg, Reg=D160, RegByteCount=1, Type=Reg, Reg=D161, RegByteCount=1

CONFIG BLOCK T_COMM K2	; Ciclo 54
  IsUserInst=false, Inst=SEND, PLCAddr=D1150, ComNum=K2, BufferCount=8, Type=Const, Data=62, RegByteCount=0, Type=Const, Data=62, RegByteCount=0, Type=Const, Data="CICLO 54", RegByteCount=0, Type=Const, Data=248, RegByteCount=0, Type=Const, Data="C", RegByteCount=0, Type=Const, Data=60, RegByteCount=0, Type=Const, Data=60, RegByteCount=0, Type=Const, Data=13, RegByteCount=0, Type=Const, Data="TEMP:", RegByteCount=0, Type=Reg, Reg=D180, RegByteCount=1, Type=Reg, Reg=D181, RegByteCount=1, Type=Reg, Reg=D182, RegByteCount=1, Type=Const, Data=248, RegByteCount=0, Type=Const, Data="C ", RegByteCount=0, Type=Const, Data="EXP:", RegByteCount=0, Type=Reg, Reg=D160, RegByteCount=1, Type=Reg, Reg=D161, RegByteCount=1, Type=Reg, Reg=D162, RegByteCount=1

CONFIG BLOCK T_COMM K3	; cada min
  IsUserInst=false, Inst=SEND, PLCAddr=D1200, ComNum=K2, BufferCount=8, Type=Const, Data="T:", RegByteCount=0, Type=Reg, Reg=D140, RegByteCount=1, Type=Reg, Reg=D141, RegByteCount=1, Type=Const, Data=".", RegByteCount=0, Type=Reg, Reg=D142, RegByteCount=1, Type=Reg, Reg=D143, RegByteCount=1, Type=Const, Data=248, RegByteCount=0, Type=Const, Data="C", RegByteCount=0, Type=Const, Data=" P:-0", RegByteCount=0, Type=Reg, Reg=D150, RegByteCount=1, Type=Const, Data=".", RegByteCount=0, Type=Reg, Reg=D151, RegByteCount=1, Type=Reg, Reg=D152, RegByteCount=1, Type=Const, Data="Bar", RegByteCount=0, Type=Const, Data=" H:", RegByteCount=0, Type=Reg, Reg=D146, RegByteCount=1, Type=Reg, Reg=D147, RegByteCount=1, Type=Const, Data="%", RegByteCount=0

CONFIG BLOCK T_COMM K4	; Condicion
  IsUserInst=false, Inst=SEND, PLCAddr=D1250, ComNum=K2, BufferCount=8, Type=Const, Data="CONDICION ", RegByteCount=0, Type=Reg, Reg=D130, RegByteCount=1, Type=Reg, Reg=D131, RegByteCount=1, Type=Const, Data=":", RegByteCount=0, Type=Reg, Reg=D132, RegByteCount=1, Type=Reg, Reg=D133, RegByteCount=1, Type=Const, Data=13, RegByteCount=0, GUID=b175af3f-664e-46ec-a7b7-4da5e1a8fe57

CONFIG BLOCK T_COMM K5	; EXPOSICION
  IsUserInst=false, Inst=SEND, PLCAddr=D1300, ComNum=K2, BufferCount=8, Type=Const, Data="EXPOSICION ", RegByteCount=0, Type=Reg, Reg=D130, RegByteCount=1, Type=Reg, Reg=D131, RegByteCount=1, Type=Const, Data=":", RegByteCount=0, Type=Reg, Reg=D132, RegByteCount=1, Type=Reg, Reg=D133, RegByteCount=1, Type=Const, Data=13, RegByteCount=0, GUID=a385d12f-5a73-4d73-8243-e5836155ab8d

CONFIG BLOCK T_COMM K6	; PURGAS
  IsUserInst=false, Inst=SEND, PLCAddr=D1350, ComNum=K2, BufferCount=8, Type=Const, Data="PURGAS ", RegByteCount=0, Type=Reg, Reg=D130, RegByteCount=1, Type=Reg, Reg=D131, RegByteCount=1, Type=Const, Data=":", RegByteCount=0, Type=Reg, Reg=D132, RegByteCount=1, Type=Reg, Reg=D133, RegByteCount=1, Type=Const, Data=13, RegByteCount=0, GUID=ea26fd37-60bd-4802-9fe9-30a961a19261

CONFIG BLOCK T_COMM K7	; AIREACION
  IsUserInst=false, Inst=SEND, PLCAddr=D1400, ComNum=K2, BufferCount=8, Type=Const, Data="AIREACION ", RegByteCount=0, Type=Reg, Reg=D130, RegByteCount=1, Type=Reg, Reg=D131, RegByteCount=1, Type=Const, Data=":", RegByteCount=0, Type=Reg, Reg=D132, RegByteCount=1, Type=Reg, Reg=D133, RegByteCount=1, Type=Const, Data=13, RegByteCount=0, GUID=36e5a285-d996-41c2-99f4-05222534c1cb

CONFIG BLOCK T_COMM K8	; ETIQUETA FIN
  IsUserInst=false, Inst=SEND, PLCAddr=D1450, ComNum=K2, BufferCount=8, Type=Const, Data="HORA FIN: ", RegByteCount=0, Type=Reg, Reg=D130, RegByteCount=1, Type=Reg, Reg=D131, RegByteCount=1, Type=Const, Data=":", RegByteCount=0, Type=Reg, Reg=D132, RegByteCount=1, Type=Reg, Reg=D133, RegByteCount=1, Type=Const, Data=":", RegByteCount=0, Type=Reg, Reg=D134, RegByteCount=1, Type=Reg, Reg=D135, RegByteCount=1, Type=Const, Data=13, RegByteCount=0, Type=Const, Data="CARGA:__________________", RegByteCount=0, Type=Const, Data=13, RegByteCount=0, Type=Const, Data="DESCARGA:_________________", RegByteCount=0, Type=Const, Data=13, RegByteCount=0, Type=Const, Data="       ", RegByteCount=0, Type=Const, Data=13, RegByteCount=0, Type=Const, Data=13, RegByteCount=0, GUID=567e5ee6-0884-405e-98a3-30450c955275

C FUNCTION BLOCK DECOFUNC.FCB
/*************************************************************************
   FunctionBlockName:  DECOFUNC
   Version:            1.0.0
   Author:             Rafael Garcia
   UpdateTime:         01/12/2016 08:27:17 a.m.
   Comment:            
			Convertir dato decimal a ascii
**************************************************************************/
void DECOFUNC( WORD W , BIT B )
{

int data, und, dec, cen, deci, data_raw, temp1, temp2;

data_raw = W[0];

data = abs(data_raw);

if (data >= 1000){
deci = data%10;
temp1 = data/10;
und = temp1%10;
temp2 = temp1/10;
dec = temp2%10;
cen = temp2/10;

W[7] = deci | 0x30;
W[6] = und | 0x30;
W[5] = dec| 0x30;
W[4] = cen | 0x30;

}

if(data >= 100 && data<1000){
und = data%10;
temp1 = data/10;
dec = temp1%10;
cen = temp1/10;

W[6] = und | 0x30;
W[5] = dec| 0x30;
W[4] = cen | 0x30;
}

if(data >= 10 && data <100 ){
und = data%10;
temp1 = data/10;
dec = temp1%10;

W[6] = und | 0x30;
W[5] = dec| 0x30;
W[4] = 00; //NULL

}

if(data >= 0 && data <10 ){
und = data%10;
temp1 = data/10;

W[6] = und | 0x30;
W[5] = 48; //cero
W[4] = 00; //NULL

}


}